// TIA Portal V16 export
// export: Created 2021-11-12T13:33:18.0098129Z, ExportSetting WithDefaults, DisplayName Totally Integrated Automation Portal, DisplayVersion V16 Update 3, DisplayName TIA Portal Version Control Interface, DisplayVersion V16 Update 2, DisplayName TIA Portal Openness, DisplayVersion V16 Update 3, DisplayName SINAMICS Startdrive Advanced, DisplayVersion V16 Update 5, DisplayName SINAMICS Startdrive G130, G150, S120, S150, SINAMICS MV, S210, DisplayVersion V16 Update 5, DisplayName SINAMICS Startdrive G110M, G120, G120C, G120D, G120P, G115D, DisplayVersion V16 Update 5, DisplayName STEP 7 Professional, DisplayVersion V16 Update 3, DisplayName STEP 7 Safety, DisplayVersion V16, DisplayName WinCC UA Professional, DisplayVersion V16 Update 3
FUNCTION_BLOCK "UserDiag_Diagnostics"   // FB21003, LAD
{ S7_Optimized_Access := 'TRUE' }
VERSION : 0.1
// //============================================================================
// //SIEMENS AG
// //(c)Copyright 2017 All Rights Reserved
// //-----------------------------------------------------------------------------
// //Library: -
// //Tested with: CPU 1214C DC/DC/DC FW4.2
// //Engineering: TIA Portal V15
// //Restrictions: -
// //Requirements: -
// //Functionality: Main FB for diagnostics
// //-----------------------------------------------------------------------------
// //Change log table:
// //Version  Date              Expert in charge                               Changes applied
// //01.00.00 25.04.2017 Siemens Industry Online Support First released version
// //01.01.00 01.12.2017 Siemens Industry Online Support Renamed in "UserDiag_Diagnostics"
// //                                                                                                    Check Flag "startDiag"
// //============================================================================
// stored: AutoNumber false, IsIECCheckEnabled false, IsRetainMemResEnabled false, MemoryReserve 100, SetENOAutomatically false, UDAEnableTagReadback false
   VAR_IN_OUT
      startDiag { ExternalAccessible := 'False'; ExternalVisible := 'False'; ExternalWritable := 'False'} : Bool;   // Startflag for diagnostic
      plcData : "UserDiag_typePLC";   // PLC diagnostics data
      ioSystemData : Array[1.."USERDIAG_IO_SYSTEMS_UPPER_LIM"] of "UserDiag_typeIOSystem";   // IO-System diagnostics data
   END_VAR
   VAR
      instPLCCheck { ExternalAccessible := 'False'; ExternalVisible := 'False'; ExternalWritable := 'False'; S7_SetPoint := 'True'} : "UserDiag_PLCCheck";   // Instance of "UserDiag_PLCCheck"
      instIOSystemCheck1 { ExternalAccessible := 'False'; ExternalVisible := 'False'; ExternalWritable := 'False'; S7_SetPoint := 'True'} : "UserDiag_IOSystemCheck";   // Instance of "UserDiag_IOSystemCheck"
      instIOSystemCheck2 { ExternalAccessible := 'False'; ExternalVisible := 'False'; ExternalWritable := 'False'; S7_SetPoint := 'True'} : "UserDiag_IOSystemCheck";   // Instance of "UserDiag_IOSystemCheck"
   END_VAR
BEGIN

REGION Network 1: Check Startflag for diagnostic
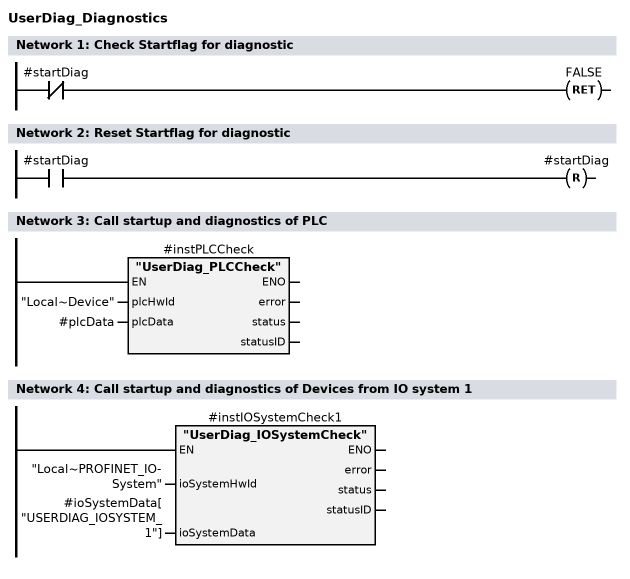
   IF NOT #startDiag THEN
       ENO := FALSE;
       RETURN;
   END_IF;
END_REGION

REGION Network 2: Reset Startflag for diagnostic
   RUNG wire#powerrail
      Contact( #startDiag )
      R_Coil( #startDiag )
   END_RUNG
   // the same network as SCL:
   IF #startDiag THEN #startDiag := FALSE; END_IF;
END_REGION

REGION Network 3: Call startup and diagnostics of PLC
   RUNG wire#powerrail
      #instPLCCheck(plcHwId := "Local~Device", plcData := #plcData, error =>, status =>, statusID =>)
   END_RUNG
   // the same network as SCL:
   #instPLCCheck(plcHwId := "Local~Device", plcData := #plcData);   // "UserDiag_PLCCheck"
END_REGION

REGION Network 4: Call startup and diagnostics of Devices from IO system 1
   RUNG wire#powerrail
      #instIOSystemCheck1(ioSystemHwId := "Local~PROFINET_IO-System", ioSystemData := #ioSystemData["USERDIAG_IOSYSTEM_1"], error =>, status =>, statusID =>)
   END_RUNG
   // the same network as SCL:
   #instIOSystemCheck1(ioSystemHwId := "Local~PROFINET_IO-System",   // "UserDiag_IOSystemCheck"
                       ioSystemData := #ioSystemData["USERDIAG_IOSYSTEM_1"]);
END_REGION
END_FUNCTION_BLOCK
